FUNCTION_BLOCK FB_System_BHKW_922
VAR_INPUT
	Freigabe_auto			: BOOL := TRUE;
	Betrieb_Anford_auto		: BOOL := FALSE;
	Regelung_Sollw_auto		: REAL := 60;
END_VAR
VAR_OUTPUT
	{attribute 'OPC.UA.DA' := '1'}Steuerung				: ST_System_BHKW_Steuerung;		
	{attribute 'OPC.UA.DA' := '1'}Stellwert					: ST_System_BHKW_Stellwert;	
	{attribute 'OPC.UA.DA' := '1'}Zustand					: ST_System_BHKW_Zustand;	
	{attribute 'OPC.UA.DA' := '1'}Parameter				: ST_System_BHKW_Parameter;		
END_VAR
VAR
	Pumpe_322				: FB_PU;
	Stellventil_322			: FB_SVs;
	Regelventil_322			: FB_RV;	(*14.07.2020*)
	BHKW_922				: FB_BHKW;

	Zustandscheck			: FB_System_BHKW_Zustandscheck;
	Logik					: FB_System_BHKW_Logik;
	Ablaufsteuerung			: FB_System_BHKW_Ablaufsteuerung;

	Timer1: TON;
	Timer_BHKW922_Pumpe322_Freigabe: 	TOF;
	Sollwertscheck: FB_System_BHKW_Sollwertscheck;
END_VAR
VAR // added by the converter: edge detectors and wires of the graphical bodies
    _w1, _w2, _w3, _w4, _w5 : ANY;
END_VAR

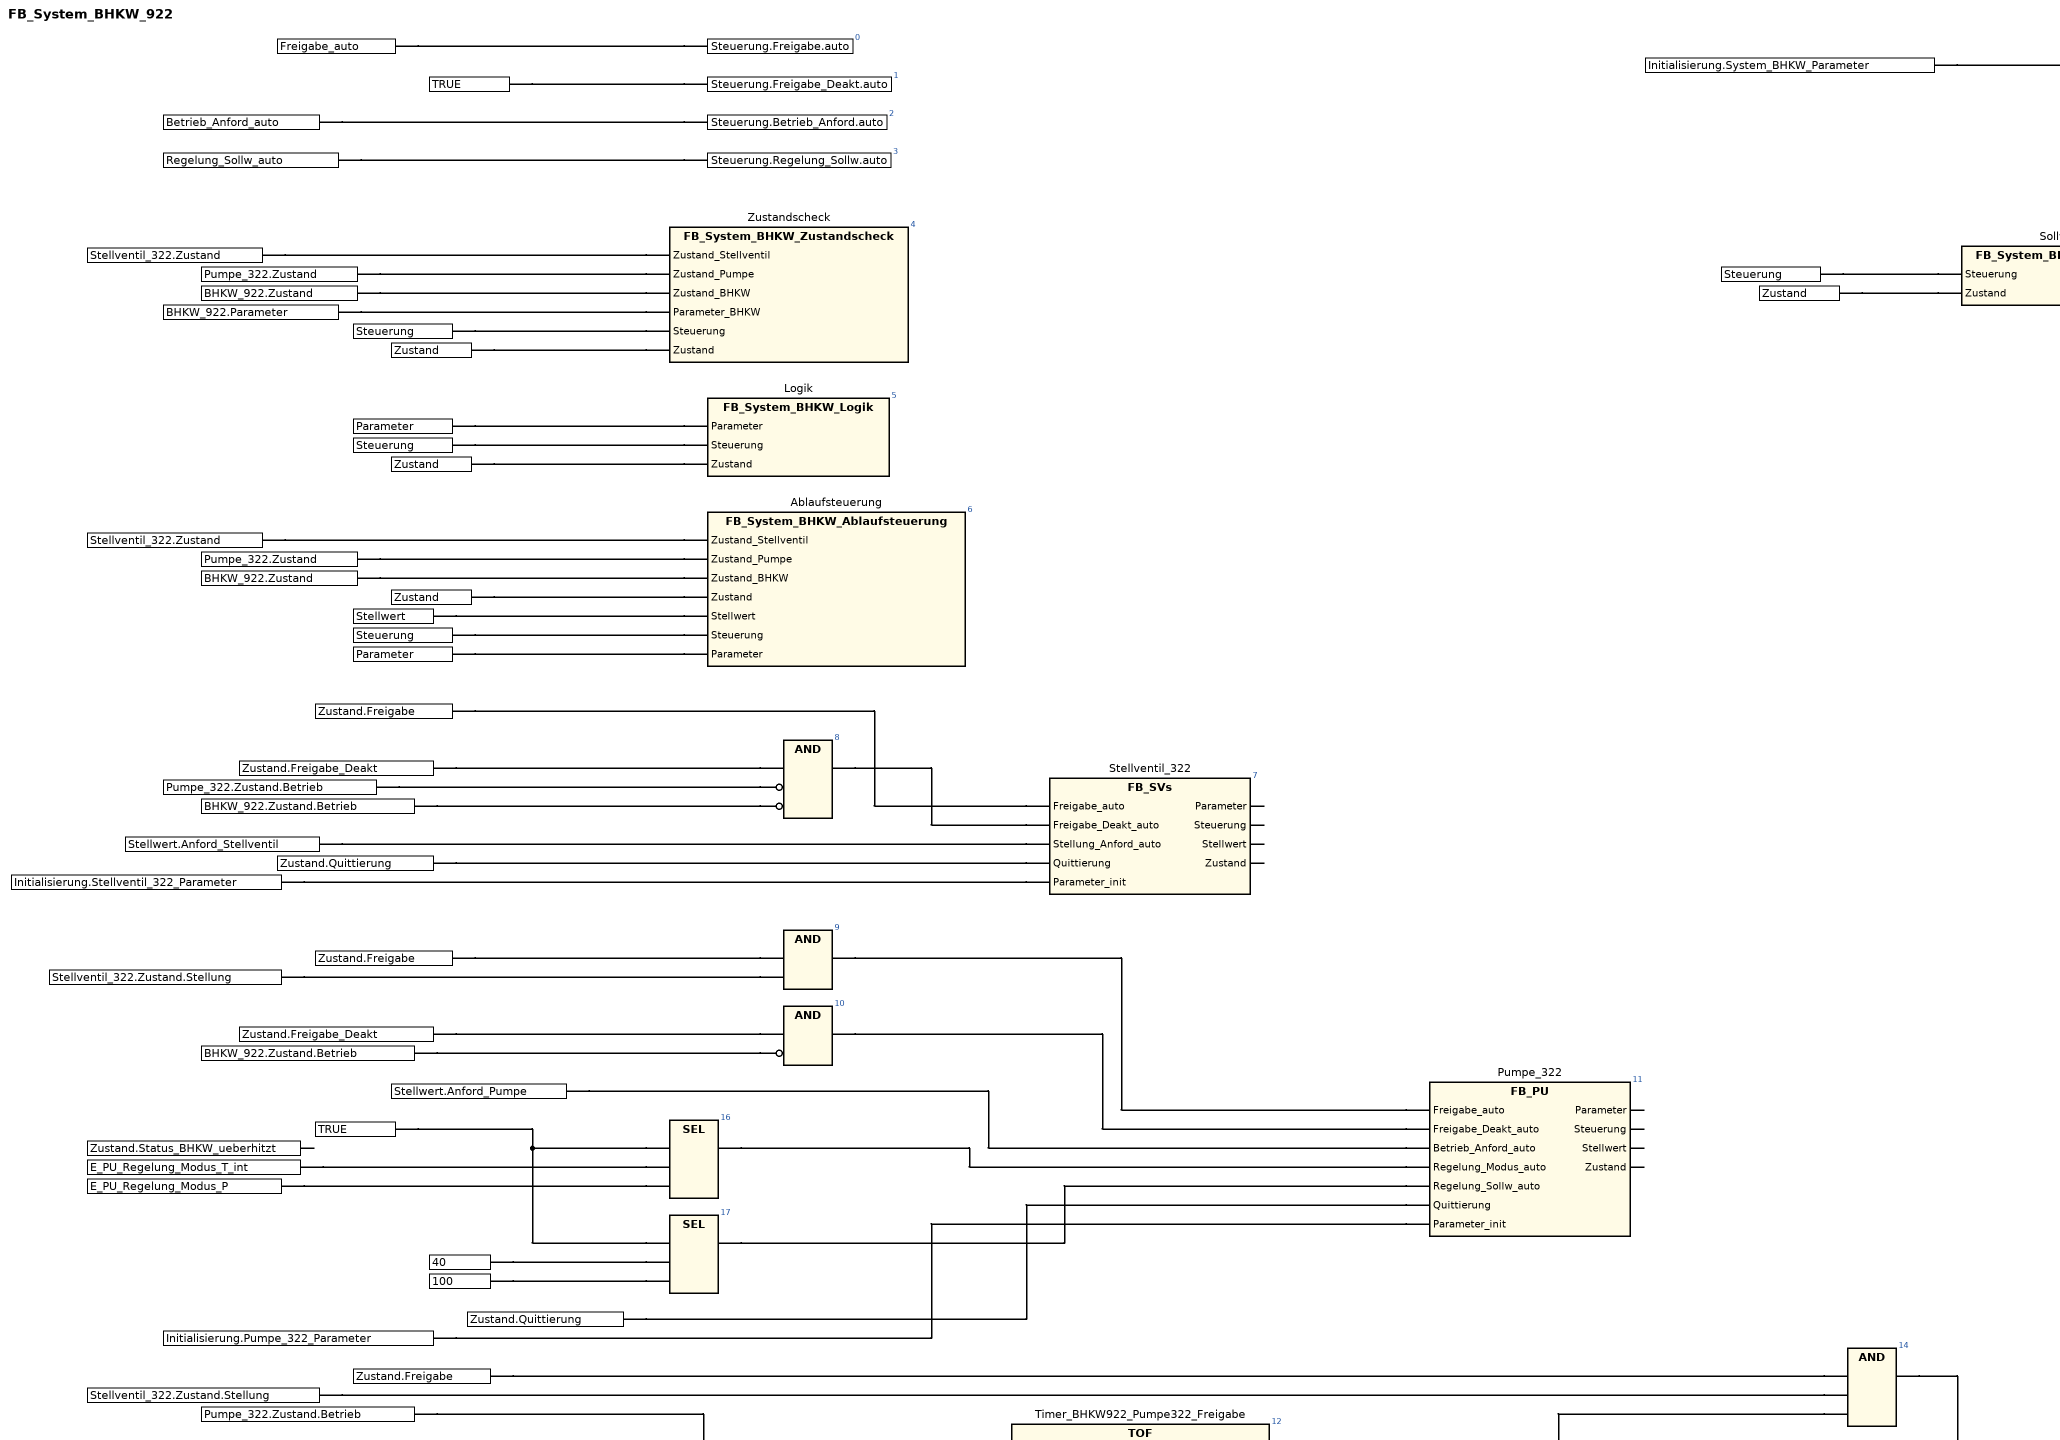
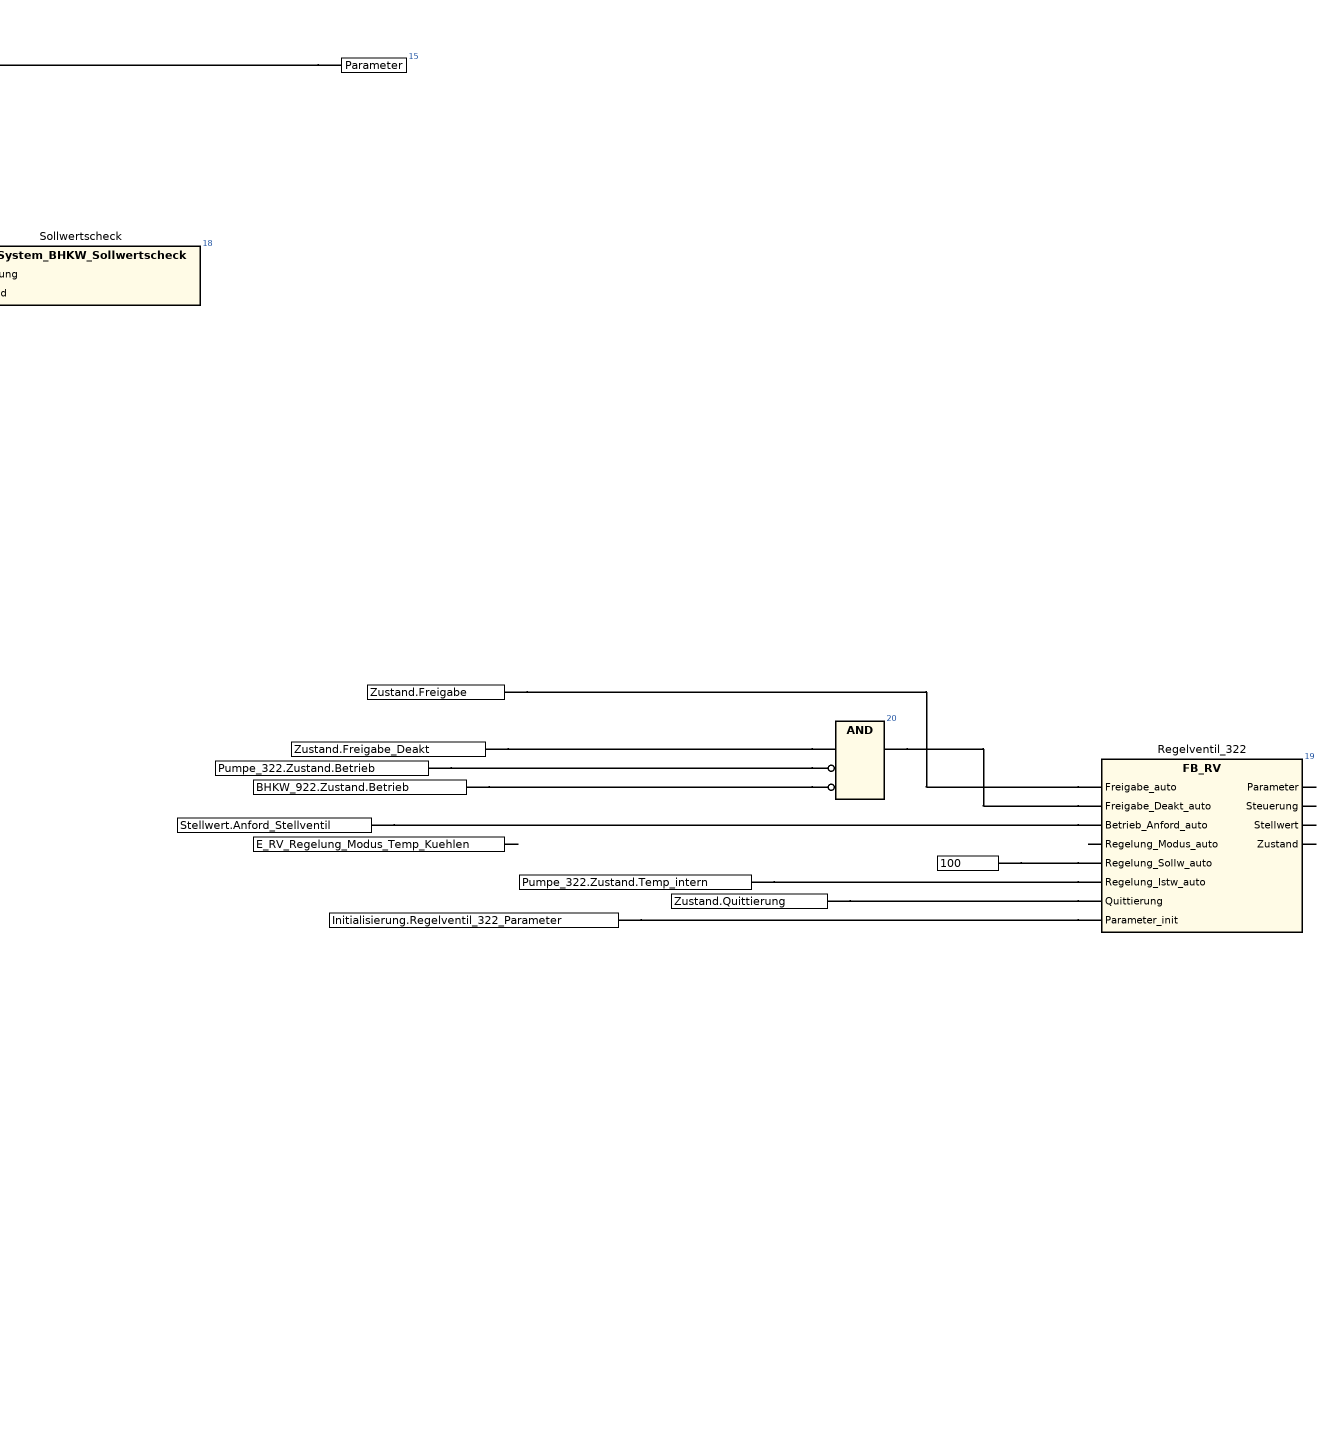
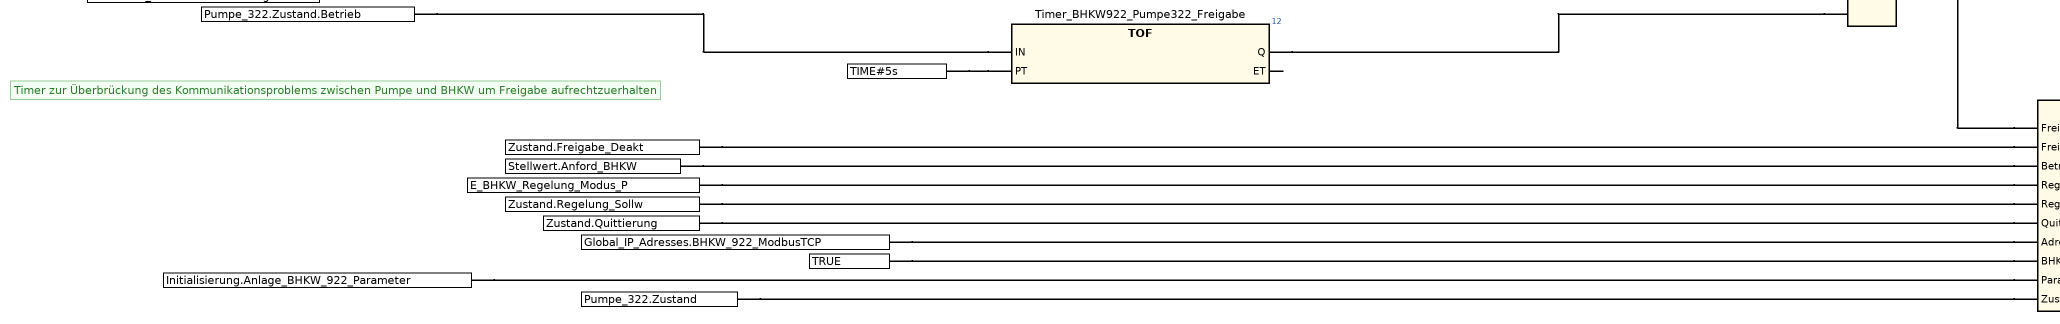
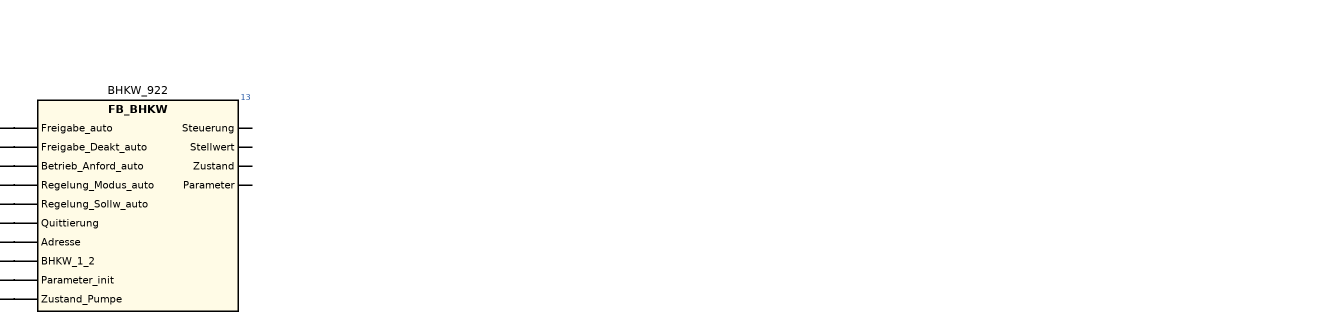
Steuerung.Freigabe.auto := Freigabe_auto;
Steuerung.Freigabe_Deakt.auto := TRUE;
Steuerung.Betrieb_Anford.auto := Betrieb_Anford_auto;
Steuerung.Regelung_Sollw.auto := Regelung_Sollw_auto;
Zustandscheck(
    Zustand_Stellventil := Stellventil_322.Zustand,
    Zustand_Pumpe := Pumpe_322.Zustand,
    Zustand_BHKW := BHKW_922.Zustand,
    Parameter_BHKW := BHKW_922.Parameter,
    Steuerung := Steuerung,
    Zustand := Zustand); // FB_System_BHKW_Zustandscheck
Logik(Parameter := Parameter, Steuerung := Steuerung, Zustand := Zustand); // FB_System_BHKW_Logik
Ablaufsteuerung(
    Zustand_Stellventil := Stellventil_322.Zustand,
    Zustand_Pumpe := Pumpe_322.Zustand,
    Zustand_BHKW := BHKW_922.Zustand,
    Zustand := Zustand,
    Stellwert := Stellwert,
    Steuerung := Steuerung,
    Parameter := Parameter); // FB_System_BHKW_Ablaufsteuerung
Stellventil_322(
    Freigabe_auto := Zustand.Freigabe,
    Freigabe_Deakt_auto := _w1,
    Stellung_Anford_auto := Stellwert.Anford_Stellventil,
    Quittierung := Zustand.Quittierung,
    Parameter_init := Initialisierung.Stellventil_322_Parameter); // FB_SVs
_w1 := Zustand.Freigabe_Deakt AND NOT Pumpe_322.Zustand.Betrieb AND NOT BHKW_922.Zustand.Betrieb;
Pumpe_322(
    Freigabe_auto := Zustand.Freigabe AND Stellventil_322.Zustand.Stellung,
    Freigabe_Deakt_auto := Zustand.Freigabe_Deakt AND NOT BHKW_922.Zustand.Betrieb,
    Betrieb_Anford_auto := Stellwert.Anford_Pumpe,
    Regelung_Modus_auto := _w2,
    Regelung_Sollw_auto := _w3,
    Quittierung := Zustand.Quittierung,
    Parameter_init := Initialisierung.Pumpe_322_Parameter); // FB_PU
// Timer zur Überbrückung des Kommunikationsproblems zwischen Pumpe und BHKW um Freigabe aufrechtzuerhalten
Timer_BHKW922_Pumpe322_Freigabe(IN := Pumpe_322.Zustand.Betrieb, PT := TIME#5s); // TOF
BHKW_922(
    Freigabe_auto := _w4,
    Freigabe_Deakt_auto := Zustand.Freigabe_Deakt,
    Betrieb_Anford_auto := Stellwert.Anford_BHKW,
    Regelung_Modus_auto := E_BHKW_Regelung_Modus_P,
    Regelung_Sollw_auto := Zustand.Regelung_Sollw,
    Quittierung := Zustand.Quittierung,
    Adresse := Global_IP_Adresses.BHKW_922_ModbusTCP,
    BHKW_1_2 := TRUE,
    Parameter_init := Initialisierung.Anlage_BHKW_922_Parameter,
    Zustand_Pumpe := Pumpe_322.Zustand); // FB_BHKW
_w4 := Zustand.Freigabe AND Stellventil_322.Zustand.Stellung AND Timer_BHKW922_Pumpe322_Freigabe.Q;
Parameter := Initialisierung.System_BHKW_Parameter;
_w2 := SEL(TRUE, E_PU_Regelung_Modus_T_int, E_PU_Regelung_Modus_P);
_w3 := SEL(TRUE, 40, 100);
Sollwertscheck(Steuerung := Steuerung, Zustand := Zustand); // FB_System_BHKW_Sollwertscheck
Regelventil_322(
    Freigabe_auto := Zustand.Freigabe,
    Freigabe_Deakt_auto := _w5,
    Betrieb_Anford_auto := Stellwert.Anford_Stellventil,
    Regelung_Sollw_auto := 100,
    Regelung_Istw_auto := Pumpe_322.Zustand.Temp_intern,
    Quittierung := Zustand.Quittierung,
    Parameter_init := Initialisierung.Regelventil_322_Parameter); // FB_RV
_w5 := Zustand.Freigabe_Deakt AND NOT Pumpe_322.Zustand.Betrieb AND NOT BHKW_922.Zustand.Betrieb;
// E_RV_Regelung_Modus_Temp_Kuehlen: input not connected
// Zustand.Status_BHKW_ueberhitzt: input not connected

END_FUNCTION_BLOCK

(* stored: Version 1.1.0.1, ProductVersion 3.1.4024.9
   POU FB_System_BHKW_922: Id {6b18ae9b-4cc8-4555-b4b8-2043e0706b2e}, SpecialFunc None *)
